(* PLC project CHL-DZ-BJDX-11 宁波数字孪生（东方理工）研究院制备薄层色谱全自动化工作站_Old_InoProShop(V1.9.1.6).project, Inovance company InoProShop(V1.9.1.6) InoProShop(V1.9.1.6) *)
(* stored: creationDateTime 2026-06-16T17:57:04.779242, modificationDateTime 2026-06-04T10:59:46 *)

ACTION A10_上下料伺服流程:
            //初始化
IF MODE_State =4 OR  初始化  THEN

		玻璃上料轴1ZDATE.fAbsTarget :=0;
		玻璃上料轴1ZDATE.xMoveAbs:=TRUE;
		玻璃上料轴1ZDATE.xJogPos :=FALSE;
		升降上料伺服允许取料 :=FALSE ;
		升降上料伺服下降完成 :=FALSE ;
		伺服上料_Setp:=0;
		伺服上料_Setp:=0;
		升降下料伺服允许放料  :=FALSE ;
		玻璃上料轴2ZDATE.xJogNeg :=FALSE;
		玻璃上料轴2ZDATE.xJogPos :=FALSE;
	
END_IF



//上料流程
IF MODE_State =1 THEN     //自动模式下
	IF 玻璃上料轴1ZDATE.bHomed AND 玻璃升降接近开关1 AND 上料进料传感器 AND 伺服上料_Setp=0 AND NOT Alarm.0 AND 升降上料完成 THEN
		伺服上料_Setp :=1;
	END_IF
	
    CASE 伺服上料_Setp OF
    	1 :
			IF NOT 玻璃升降光电开关1 AND 玻璃上料轴1ZDATE.fActPos<514  THEN
				Z1JOG_pos :=TRUE;
				ELSE
				Z1JOG_pos :=FALSE;
				伺服上料_Setp:=10;
			END_IF
   
	   10:
		   IF 玻璃升降光电开关1 THEN
		   	升降上料伺服允许取料 :=TRUE;
			伺服上料_Setp:=20;
		   END_IF
		   
	   20:
		   IF 升降上料机器人已吸住物料 THEN
		   	玻璃上料轴1ZDATE.fRelTarget :=-5.0;
			玻璃上料轴1ZDATE.xMoveRel :=TRUE;
			伺服上料_Setp:=30;
		   END_IF
	   30:
		   IF 玻璃上料轴1ZDATE .bReMoveDone  THEN
		   	升降上料伺服下降完成 :=TRUE ;
			玻璃上料轴1ZDATE.xMoveRel :=FALSE;
			伺服上料_Setp:=40;
		   END_IF
	   40:
		   IF 升降上料机器人取料完成  THEN
		   	升降上料伺服下降完成 :=FALSE ;
			升降上料伺服允许取料 :=FALSE ;
			伺服上料_Setp:=1;
		   END_IF 
    END_CASE
	
	IF 玻璃上料轴1ZDATE.fActPos>=514 AND  玻璃升降光电开关1 THEN
		Alarm.0:=TRUE;                                             //上料机构无物料
		升降上料完成:=FALSE;
		玻璃上料轴1ZDATE.fAbsTarget :=0;
		玻璃上料轴1ZDATE.xMoveAbs:=TRUE;
		Z1JOG_pos :=FALSE;
		升降上料伺服允许取料 :=FALSE ;
		升降上料伺服下降完成 :=FALSE ;
		伺服上料_Setp:=0;
	END_IF
	IF 玻璃上料轴1ZDATE .bAbMoveDone  THEN
		玻璃上料轴1ZDATE.xMoveAbs:=FALSE;
		升降上料机器人放料完成:=FALSE;
    END_IF
	
	
END_IF
//下料流程
IF MODE_State =1 THEN     //自动模式下
	IF 玻璃上料轴2ZDATE.bHomed  AND 下料出料传感器 AND 伺服下料_Setp=0 AND NOT Alarm.1 AND 升降下料完成 THEN
		伺服下料_Setp :=1;
	END_IF
	
    CASE 伺服下料_Setp  OF
    	1 :
			IF NOT 玻璃升降光电开关2 AND 玻璃上料轴2ZDATE.fActPos<510  THEN
				Z2JOG_POS :=TRUE;
				ELSE
				Z2JOG_POS :=FALSE;
				伺服下料_Setp:=10;
			END_IF
   
	   10:
		   IF 玻璃升降光电开关2 THEN
			   Z2JOG_NEG :=TRUE;
			   伺服下料_Setp:=15;
		   END_IF
	   15:
		   IF NOT 玻璃升降光电开关2  THEN
				升降下料伺服允许放料  :=TRUE;
				Z2JOG_NEG :=FALSE;
				伺服下料_Setp:=20;
		   END_IF
			  
	   
	   20:
		   IF 升降下料机器人放废料完成 AND 玻璃升降光电开关2 AND 玻璃升降接近开关2 THEN
		   	Z2JOG_NEG :=TRUE;
			升降下料伺服允许放料  :=FALSE ;
			伺服下料_Setp:=30;
		   END_IF
		  
	   30:
		   IF NOT 玻璃升降光电开关2 THEN
		   	Z2JOG_NEG :=FALSE;
			伺服下料_Setp:=10;
		   END_IF
	  
    END_CASE
	
	IF 玻璃上料轴2ZDATE.fActPos<=0 AND 玻璃升降光电开关1 THEN
		Alarm.1:=TRUE;                                           //下料机构已满料
		升降下料完成:=FALSE;
		伺服下料_Setp:=0;
		升降下料伺服允许放料  :=FALSE ;
		Z2JOG_NEG :=FALSE;
		Z2JOG_POS :=FALSE;
		玻璃上料轴2ZDATE.fAbsTarget :=0;
		玻璃上料轴2ZDATE.xMoveAbs:=TRUE;
		伺服下料_Setp:=0;
	END_IF
	IF 玻璃上料轴2ZDATE .bAbMoveDone  THEN
		玻璃上料轴2ZDATE.xMoveAbs:=FALSE;
		升降下料伺服允许放料  :=FALSE ;
    END_IF
END_IF















          
END_ACTION

ACTION A00_设备状态显示及控制:
            //PLC模式切换
PLC_Mode_0(
    bWarning_alarm := cyinderAlarm<>0 OR Alarm<>0 OR 上样料架报警, 

	xStart:= 启动 , 
	xStop:=NOT  停止 , 
	xReset:=复位  , 
	xAutoMode:=手自动  , 
	xFault:=伺服报警 OR ECAT掉站报警 OR 伺服未回原点报警, 
	xEmergency:= 急停 , 
	bRed=>三色灯红  , 
	bYellow=> 三色灯黄, 
	bGreen=> 三色灯绿, 
	bBuzzer=> 蜂鸣器 , 
	iState=>MODE_STATE  , 
	bAuto=>ManualAuto  );
	
	//伺服报错
IF   玻璃上料轴1ZDATE.bError OR 玻璃上料轴2ZDATE.bError OR 打样瓶上料轴3YDATE.bError OR 点样轴6XDATE.bError OR 点样轴7YDATE.bError OR 拍照轴8YDATE.bError OR 刮板轴9XDATE.bError OR 刮板轴10ZDATE.bError OR 地轨轴11YDATE.bError OR 上样轴4X轴DATE.bError OR 上样轴5Z轴DATE.bError THEN
	伺服报警:=TRUE;
END_IF
   //伺服报错复位
IF 复位 THEN
	伺服报警:=FALSE;
	伺服未回原点报警:=FALSE;
	Alarm:=0;
	cyinderAlarm:=0;
	上样料架报警:=FALSE;
END_IF


IF NOT 玻璃上料轴1ZDATE.bHomed OR NOT 玻璃上料轴2ZDATE.bHomed OR NOT 打样瓶上料轴3YDATE.bHomed OR NOT 点样轴6XDATE.bHomed OR NOT 点样轴7YDATE.bHomed OR NOT 拍照轴8YDATE.bHomed OR NOT 刮板轴9XDATE.bHomed OR NOT 刮板轴10ZDATE.bHomed  OR NOT 地轨轴11YDATE.bHomed OR NOT 上样轴4X轴DATE.bHomed OR NOT 上样轴5Z轴DATE.bHomed THEN
	伺服未回原点报警:=TRUE ;
END_IF
          
END_ACTION

ACTION A20_机器人:
            //机器人远程控制
RB_Control_0(
	StartButton:=MODE_State=1 , 
	StopButton:= 初始化, 
	PulseButton:= 停止 AND NOT 急停, 
	ContinueButton:=启动 , 
	ResettButton:=复位 , 
	Ready:= RB_远程模式, 
	Running:=RB_运行中 , 
	Paused:= RB_暂停中, 
	Error:=RB_报警中 , 
	MotorOnOutput=> RB_上电, 
	StartOutput=>RB_启动 , 
	StopOutput=>RB_停止 , 
	PauseOutput=> RB_暂停, 
	ContinueOutput=> RB_继续, 
	ResetOutput=>RB_复位 );
          
END_ACTION

ACTION A30_急停:
            
伺服上料_Setp:=0;
伺服下料_Setp:=0;
//收集工位
收集下压气缸手动:=FALSE;
收集下压气缸自动:=FALSE;
收集夹持气缸手动:=FALSE;
收集夹持气缸自动:=FALSE;
收集升降气缸手动:=FALSE;
收集升降气缸自动:=FALSE;
收集伸缩气缸手动:=FALSE;
收集伸缩气缸自动:=FALSE;
收集进液手动:=FALSE;
收集进液自动:=FALSE;
收集排液手动:=FALSE;
收集排液自动:=FALSE;
收集正压排液手动:=FALSE;
收集正压排液自动:=FALSE;
溶液收集瓶定位手动:=FALSE;
收集工位允许放收集瓶:=FALSE;
收集工位允许放收集器:=FALSE;
收集工位允许机器人退出工位:=FALSE;
收集工位允许机器人取收集瓶放暂存工位:=FALSE;
收集工位允许取收集器:=FALSE;
收集工位机器人取收集器放回暂存工位:=FALSE;
collect_prepare_OK:=FALSE;
collect_OK:=FALSE;
收集工位放收集器完成:=FALSE;
//展开工位
expand_initialization_OK:=FALSE;
Expand_Group_clean_OK:=FALSE;
Expand_up_liquid_OK:=FALSE;
Expand_silica_gel_plate_OK:=FALSE;
展缸1气缸1手动:=FALSE;
展缸1气缸1自动:=FALSE;
展缸1进液电池阀1手动:=FALSE;
展缸1进液电池阀1自动:=FALSE;
展缸1排液电池阀1手动:=FALSE;
展缸1排液电池阀1自动:=FALSE;
展缸1吹气电池阀1手动:=FALSE;
展缸1吹气电池阀1自动:=FALSE;
展缸1气缸2手动:=FALSE;
展缸1气缸2自动:=FALSE;
展缸1进液电池阀2手动:=FALSE;
展缸1进液电池阀2自动:=FALSE;
展缸1排液电池阀2手动:=FALSE;
展缸1排液电池阀2自动:=FALSE;
展缸1吹气电池阀2手动:=FALSE;
展缸1吹气电池阀2自动:=FALSE;
展缸1气缸3手动:=FALSE;
展缸1气缸3自动:=FALSE;
展缸1进液电池阀3手动:=FALSE;
展缸1进液电池阀3自动:=FALSE;	
展缸1排液电池阀3手动:=FALSE;
展缸1排液电池阀3自动:=FALSE;
展缸1吹气电池阀3手动:=FALSE;
展缸1吹气电池阀3自动:=FALSE;
展缸1气缸4手动:=FALSE;
展缸1气缸4自动:=FALSE;
展缸1进液电池阀4手动:=FALSE;
展缸1进液电池阀4自动:=FALSE;	
展缸1排液电池阀4手动:=FALSE;
展缸1排液电池阀4自动:=FALSE;
展缸1吹气电池阀4手动:=FALSE;
展缸1吹气电池阀4自动:=FALSE;
展缸2气缸1手动:=FALSE;
展缸2气缸1自动:=FALSE;
展缸2进液电池阀1手动:=FALSE;
展缸2进液电池阀1自动:=FALSE;
展缸2排液电池阀1手动:=FALSE;
展缸2排液电池阀1自动:=FALSE;
展缸2吹气电池阀1手动:=FALSE;
展缸2吹气电池阀1自动:=FALSE;
展缸2气缸2手动:=FALSE;
展缸2气缸2自动:=FALSE;
展缸2进液电池阀2手动:=FALSE;
展缸2进液电池阀2自动:=FALSE;
展缸2排液电池阀2手动:=FALSE;
展缸2排液电池阀2自动:=FALSE;
展缸2吹气电池阀2手动:=FALSE;
展缸2吹气电池阀2自动:=FALSE;
展缸2气缸3手动:=FALSE;
展缸2气缸3自动:=FALSE;
展缸2进液电池阀3手动:=FALSE;
展缸2进液电池阀3自动:=FALSE;	
展缸2排液电池阀3手动:=FALSE;
展缸2排液电池阀3自动:=FALSE;
展缸2吹气电池阀3手动:=FALSE;
展缸2吹气电池阀3自动:=FALSE;
展缸2气缸4手动:=FALSE;
展缸2气缸4自动:=FALSE;
展缸2进液电池阀4手动:=FALSE;
展缸2进液电池阀4自动:=FALSE;	
展缸2排液电池阀4手动:=FALSE;
展缸2排液电池阀4自动:=FALSE;
展缸2吹气电池阀4手动:=FALSE;
展缸2吹气电池阀4自动:=FALSE;
//拍照刮板
刮板拍照真空自动:=FALSE;
刮板拍照真空手动:=FALSE;
刮板拍照无刷电机手动:=FALSE;
刮板拍照无刷电机自动:=FALSE;
刮板拍照定位气缸手动:=FALSE;
刮板拍照定位气缸自动:=FALSE;
粉末收集器定位手动:=FALSE;
粉末收集器定位自动:=FALSE;
刮板拍照遮光气缸手动:=FALSE;
刮板拍照遮光气缸自动:=FALSE;
刮板拍照旋转气缸手动:=FALSE;
刮板拍照旋转气缸自动:=FALSE;
刮板拍照下压气缸手动:=FALSE;
刮板拍照下压气缸自动:=FALSE;
拍照工位允许放硅胶板:=FALSE;
拍照工位允许放收集器:=FALSE;
拍照工位机器人退出工位:=FALSE;
拍照工位允许取收集器:=FALSE;
拍照工位机器人退出:=FALSE;
scrape_WaitConfirm := FALSE;
Camera_scraper_initialization_OK:=FALSE;
Photo_preparation_completed_OK:=FALSE;
Scraper_collection_completed:=FALSE;
Robot_completes_material_retrieval:=FALSE;		
//上样点样
上样定位手动:=FALSE;
上样定位自动:=FALSE;
上样点样三通电池阀手动:=FALSE;
上样点样三通电池阀自动:=FALSE;
上样吹气手动:=FALSE;
上样吹气自动:=FALSE;
打样瓶上料轴3YDATE.fAbsTarget:=0;
点样轴6XDATE.fAbsTarget:=0;
点样轴7YDATE.fAbsTarget:=0;
上样轴4X轴DATE.fAbsTarget:=0;
上样轴5Z轴DATE.fAbsTarget:=0;
上样点样允许放硅胶板:=FALSE;
点样轴7YDATE.xMoveAbs:=FALSE;
点样轴6XDATE.xMoveAbs:=FALSE;
上样轴5Z轴DATE.xMoveAbs:=TRUE;
上样轴4X轴DATE.xMoveAbs:=FALSE;
打样瓶上料轴3YDATE.xMoveAbs:=FALSE;
Sampling_Spray_sample_OK:=FALSE;
Sampling_liquid_absorption:=FALSE;
Sampling_preparation_OK:=FALSE;
//机器人
Execute:=0;
FunctionID:=0;
ParameterList1:=0;
ParameterList2:=0;
ParameterList3:=0;
ParameterList4:=0;
ParameterList5:=0;
ParameterList6:=0;
ParameterList7:=0;
ParameterList8:=0;
ParameterList9:=0;
ParameterList10:=0;




上样料架报警:=FALSE;
取工具setp:=0;
取工具完成:=FALSE;
取升降硅胶板step:=0;
取升降硅胶板完成:=FALSE;
放点样硅胶板step:=0;
放点样硅胶板完成:=FALSE;
取点样硅胶板step:=0;
取点样硅胶板完成:=FALSE;
放展缸硅胶板完成:=FALSE;
放展缸硅胶板step:=0;
取展缸硅胶板step:=0;
取展缸硅胶板完成:=FALSE;
放拍照硅胶板完成:=FALSE;
放拍照硅胶板step:=0;
取收集器组放暂存工位step:=0;
取收集瓶组放暂存工位完成:=FALSE;
取暂存收集器放刮板位完成:=FALSE;
取暂存收集器放刮板位step:=0;
取刮板收集器放到收集工位完成:=FALSE;
取刮板收集器放到收集工位step:=0;
取暂存收集瓶放收集工位step:=0;
取暂存收集瓶放收集工位完成:=FALSE;
取收集器放暂存工位完成:=FALSE;
取收集器放暂存工位step:=0;
取刮板硅胶板放废料区step:=0;
取刮板硅胶板放废料区完成:=FALSE;
取暂存收集器组放仓库完成:=FALSE;
取暂存收集器组放仓库step:=0;
取收集器组放暂存工位完成:=FALSE;
取收集瓶组放暂存工位step:=0;
取暂存收集瓶组放仓库完成:=FALSE;
取暂存收集瓶组放仓库step:=0;
取收集瓶放暂存工位step:=0;
取收集瓶放暂存工位完成:=FALSE;

          
END_ACTION

PROGRAM PLC_MainPRG
  VAR
    PLC_Mode_0 : FB_Mode;
    TON_1 : TON;
    RB_Control_0 : FB_RB_Control;
    TON_0 : TON;
    TON_2 : TON;
    TON_3 : TON;
    SysHC_ModbusTcpSlaveDiagnose_0 : SysHC_ModbusTcpSlaveDiagnose;
  END_VAR

            
A00_设备状态显示及控制 ();

A20_机器人();
%MW1000:=0;

PLC_Cyinder_气缸动作();

CASE MODE_State OF
	EN_功能块状态.运行:
		A10_上下料伺服流程 ();
		Sample_point_sampling_上样点样();
		Collection_process_收集流程();
		Expand_process_展开流程();
		Photo_scraper_拍照刮板();
		Robotic_Process_机器人流程();
		Develop_TankDrain();
		
END_CASE

TON_3(IN:=复位,PT:=T#5S );
IF NOT 急停 OR TON_3.Q THEN
	A30_急停();
END_IF
IF MODE_State<>1 THEN
	伺服上料_Setp:=0;
	伺服下料_Setp:=0;
END_IF



          
END_PROGRAM
